DATA_BLOCK "DB_Integers"
{ S7_Optimized_Access := 'TRUE' }
VERSION : 0.1
NON_RETAIN
   VAR
      Int_Min_n32768 : Int;   // Int: Min
      Int_Max_32767 : Int;   // Int: Max
      Int_12345 : Int;   // Int: Testvalue 1
      Int_n9876 : Int;   // Int: Testvalue 2
      Int_write : Int;   // Write test
      ULInt_Min_0 : ULInt;   // ULInt: Min
      ULInt_Max_18446744073709551615 : ULInt;   // ULInt: Max
      ULInt_12345678901234567890 : ULInt;   // ULInt: Testvalue 1
      ULInt_write : ULInt;   // Write test
      LInt_Min_n9223372036854775808 : LInt;   // LInt: Min
      LInt_Max_9223372036854775807 : LInt;   // LInt: Max
      LInt_1234567890123456789 : LInt;   // LInt: Testvalue 1
      LInt_n987654321098765432 : LInt;   // LInt: Testvalue 2
      LInt_write : LInt;   // Write test
      USint_Min_0 : USInt;   // USInt: Min
      USInt_Max_255 : USInt;   // USInt: Max
      USInt_123 : USInt;   // USInt: Testvalue 1
      USInt_write : USInt;   // Write test
      UInt_Min_0 : UInt;   // UInt: Min
      UInt_Max_65535 : UInt;   // UInt: Max
      UInt_12345 : UInt;   // UInt: Testvalue 1
      UInt_write : UInt;   // Write test
      UDInt_Min_0 : UDInt;   // UDInt: Min
      UDInt_Max_4294967295 : UDInt;   // UDInt: Max
      UDint_1234567890 : UDInt;   // UDInt: Testvalue 1
      UDInt_write : UDInt;   // Write test
      SInt_Min_n128 : SInt;   // SInt: Min
      SInt_Max_127 : SInt;   // SInt: Max
      SInt_123 : SInt;   // SInt: Testvalue 1
      SInt_n123 : SInt;   // SInt: Testvalue 2
      SInt_write : SInt;   // Write test
      DInt_Min_n2147483648 : DInt;   // DInt: Min
      DInt_Max_2147483647 : DInt;   // DInt: Max
      DInt_1234567890 : DInt;   // DInt: Testvalue 1
      DInt_n987654321 : DInt;   // DInt: Testvalue 2
      DInt_write : DInt;   // Write test
   END_VAR


BEGIN
   Int_Min_n32768 := -32768;
   Int_Max_32767 := 32767;
   Int_12345 := 12345;
   Int_n9876 := -9876;
   ULInt_Max_18446744073709551615 := 18_446_744_073_709_551_615;
   ULInt_12345678901234567890 := 12_345_678_901_234_567_890;
   LInt_Min_n9223372036854775808 := -9_223_372_036_854_775_808;
   LInt_Max_9223372036854775807 := 9_223_372_036_854_775_807;
   LInt_1234567890123456789 := 1_234_567_890_123_456_789;
   LInt_n987654321098765432 := -987_654_321_098_765_432;
   USInt_Max_255 := 255;
   USInt_123 := 123;
   UInt_Max_65535 := 65535;
   UInt_12345 := 12345;
   UDInt_Max_4294967295 := 4_294_967_295;
   UDint_1234567890 := 1_234_567_890;
   SInt_Min_n128 := -128;
   SInt_Max_127 := 127;
   SInt_123 := 123;
   SInt_n123 := -123;
   DInt_Min_n2147483648 := -2_147_483_648;
   DInt_Max_2147483647 := 2_147_483_647;
   DInt_1234567890 := 1_234_567_890;
   DInt_n987654321 := -987_654_321;

END_DATA_BLOCK

